Staubli VAL3: calcTool4pEn.dtx

num nYPosButTxt = 13
num nXPosButTxt[9]
  [2] = 5
  [3] = 10
  [4] = 15
  [5] = 20
  [6] = 25
  [7] = 30
  [8] = 35
num nToolZ = 85.675524
num nToolY = 78.070962
num nToolX = 77.131006
num nScZ = -66.099092
num nScY = 338.426123
num nScX = 51.350106
num nS4[4]
  [1] = 61.687518
  [2] = 361.744122
  [3] = 70.795403
num nS3[4]
  [1] = -35.244781
  [2] = 252.515203
  [3] = 1.067367
num nS2[4]
  [1] = 154.512491
  [2] = 254.102853
  [3] = -25.629323
num nS1[4]
  [1] = 62.978505
  [2] = 253.490247
  [3] = 43.634089
num nLangSet = 100
string sUsrMess[140]
  [0] = "Please select a Language"
  [1] = "Programm zur Toolberechnung"
  [2] = "Dieses Prog. errechnet anhand 4 POINTS,"
  [3] = "die kugelfoermig um einen gemeinsamen"
  [4] = "Mittelpkt angeordnet sind,die X, Y und"
  [5] = "Z-Werte des akt. Tools. Diese Points"
  [6] = "muessen geometrisch unabhaengig sein."
  [7] = "D.h. sie duerfen nicht in EINER"
  [8] = "gemeinsamen Ebene liegen !!!"
  [9] = "Teachen der Locations !"
  [10] = "Punkt aufnehmen "
  [11] = "Aufnahme des "
  [12] = ".Punkts"
  [13] = "-Here- druecken um Punkt zu speichern"
  [14] = "ABBRUCH"
  [15] = "VORGANG ABGEBROCHEN !!!"
  [16] = ".Punkt aufgenommen !!!"
  [17] = "Mitte"
  [18] = "gemittelt"
  [19] = "Gemitteltes Tool sofort setzten ?"
  [20] = "TOOL NICHT GESETZT !!!"
  [21] = "TOOL GESETZT !!!"
  [22] = "Abbrechen       "
  [23] = "Wollen Sie fortfahren ? "
  [24] = " JA"
  [25] = "NEIN"
  [26] = "Here"
  [27] = "Ergebnis der Toolberechnung"
  [28] = "Tool-X"
  [29] = "Tool-Y"
  [30] = "Tool-Z"
  [31] = "Gemitteltes Tool => TRSF user_tool"
  [32] = "Division durch 0 nicht moeglich !!!"
  [101] = ">>  TEACH TCP:  4-Pnt Method  <<"
  [102] = "Teach new TCP by moving EOAT"
  [103] = "to Cell Ref Pntr at 4 unique locs"
  [105] = "Creates X, Y, & Z tool values ONLY."
  [109] = "MOVE EOAT to Cell Ref 4 Times"
  [110] = "Teaching Location"
  [111] = "Ready to teach Point #"
  [112] = " of 4 Points"
  [113] = "To RECORD the Point press OK"
  [114] = "ABORT"
  [115] = "PROGRAM ABORTED !"
  [116] = ".Point taught !"
  [117] = "Center"
  [118] = "average"
  [119] = "Do you want to SET average Tool now ?"
  [120] = "TOOL NOT SET !"
  [121] = "TOOL SET !"
  [122] = "ABORT"
  [123] = "  CONTINUE?"
  [124] = "YES"
  [125] = " NO"
  [126] = " OK"
  [127] = "Result of the Tool calculation"
  [128] = "Tool-X"
  [129] = "Tool-Y"
  [130] = "Tool-Z"
  [131] = "Average Tool => TRSF user_tool"
  [132] = "Division though 0 is not possible !"
bool bAbort
public trsf trUserTool = {x=77.131006, y=78.070962, z=85.675524}
trsf trCenter = {x=51.350106, y=338.426123, z=-66.099092}
trsf trTempTool[4]
  [0] = {x=77.155685, y=77.510686, z=86.196215, rx=90.377616, ry=-46.104748, rz=-5.94567}
  [1] = {x=75.398979, y=79.568198, z=85.87543, rx=-72.453473, ry=-72.098018, rz=-166.490924}
  [2] = {x=79.630974, y=75.319211, z=85.887242, rx=96.053335, ry=11.032315, rz=-5.348165}
  [3] = {x=76.338385, y=79.885751, z=84.743209, rx=148.815528, ry=-36.859344, rz=7.461805}
trsf trSphere[4]
  [0] = {x=62.978505, y=253.490247, z=43.634089, rx=-90.263366, ry=-6.21772, rz=46.076845}
  [1] = {x=154.512491, y=254.102853, z=-25.629323, rx=-84.674218, ry=-3.222629, rz=107.419069}
  [2] = {x=-35.244781, y=252.515203, z=1.067367, rx=-95.956833, ry=-4.163092, rz=-11.526641}
  [3] = {x=61.687518, y=361.744122, z=70.795403, rx=-139.721556, ry=-26.205204, rz=27.844784}
pointRx pTempS[5]
  [0] = {fatherId=world[0]}
  [1] = {x=62.978505, y=253.490247, z=43.634089, rx=-90.263366, ry=-6.21772, rz=46.076845, shoulder=lefty, elbow=epositive, wrist=wnegative, fatherId=world[0]}
  [2] = {x=154.512491, y=254.102853, z=-25.629323, rx=-84.674218, ry=-3.222629, rz=107.419069, shoulder=lefty, elbow=epositive, wrist=wnegative, fatherId=world[0]}
  [3] = {x=-35.244781, y=252.515203, z=1.067367, rx=-95.956833, ry=-4.163092, rz=-11.526641, shoulder=lefty, elbow=epositive, wrist=wnegative, fatherId=world[0]}
  [4] = {x=61.687518, y=361.744122, z=70.795403, rx=-139.721556, ry=-26.205204, rz=27.844784, shoulder=lefty, elbow=epositive, wrist=wnegative, fatherId=world[0]}
